FUNCTION CheckDivLInt : LINT
VAR_INPUT
	divisor:LINT;
END_VAR

{noflow}
IF divisor = 0 THEN
	CheckDivLInt:=1;
	oaksGVL.udiCheckDivLInt := oaksGVL.udiCheckDivLInt + 1;	
ELSE
	CheckDivLInt:=divisor;
END_IF;
{flow}

END_FUNCTION

(* stored: Version 1.1.0.1, ProductVersion 3.1.4022.18
   POU CheckDivLInt: Id {9db65794-6fa7-43be-a273-27f8cf614584}, SpecialFunc CheckDivInt64 *)
